(* IEC 61131-3 sources: jiepp/tests/jiepp/input, 3 files *)

(* ---- boost.iec ---- *)
{#include './boost/preprocessor/library.hpp'}
///{#include <boost/preprocessor/repetition/repeat.hpp>}
///{#include './boost/preprocessor/config/config.hpp'}

{#define DEFINE_IN_VAR(z, n, data) BOOST_PP_CAT(in, BOOST_PP_ADD(n, 1)): data;}
{#define SUM_IN_VARS(z, n, data) BOOST_PP_IF(n, +, ) BOOST_PP_CAT(in, BOOST_PP_ADD(n, 1))}

{#define DEFINE_ADD_FUNCTION(z, n, data) $
function BOOST_PP_CAT(add_, BOOST_PP_CAT(BOOST_PP_CAT(data, _), BOOST_PP_ADD(n, 2))): data $
var_input $
    BOOST_PP_REPEAT(BOOST_PP_ADD(n, 2), DEFINE_IN_VAR, data) $
end_var $
$
BOOST_PP_CAT(add_, BOOST_PP_CAT(BOOST_PP_CAT(data, _), BOOST_PP_ADD(n, 2))) := BOOST_PP_REPEAT(BOOST_PP_ADD(n, 2), SUM_IN_VARS, _); $
$
end_function $
}

BOOST_PP_REPEAT(8, DEFINE_ADD_FUNCTION, int)

{#undef SUM_IN_VARS}
{#undef DEFINE_IN_VAR}

(* ---- function_macro.iec ---- *)
{#define DECL_BIN_FUNCTION(PREFIX, OPERATOR, T) $
function PREFIX@@_@@T: T $
var_input $
	in1, in2: T; $
end_var $
$
PREFIX@@_@@T := in1 OPERATOR in2; $
$
end_function}

{#define DECL_ADD_FUNCTION(T) DECL_BIN_FUNCTION(add, +, T)}
{#define DECL_MUL_FUNCTION(T) DECL_BIN_FUNCTION(mul, *, T)}

DECL_ADD_FUNCTION(int);
DECL_MUL_FUNCTION(int);

DECL_ADD_FUNCTION(lreal);
DECL_MUL_FUNCTION(lreal);

(* ---- if.iec ---- *)
{#if true}
program Main1 __LINE__;end_program
{#endif}

{#if false}
program Main2 __LINE__;end_program
{#endif}

{#if true}
program Main3_1 __LINE__;end_program
{#else}
program Main3_2 __LINE__;end_program
{#endif}

{#if false}
program Main4_1 __LINE__;end_program
{#else}
program Main4_2 __LINE__;end_program
{#endif}

{#if false}
program Main5_1 __LINE__;end_program
{#elif false}
program Main5_2 __LINE__;end_program
{#else}
program Main5_3 __LINE__;end_program
{#endif}

{#if false}
program Main6_1 __LINE__;end_program
{#elif true}
program Main6_2 __LINE__;end_program
{#else}
program Main6_3 __LINE__;end_program
{#endif}

{#if true}
program Main7_1 __LINE__;end_program
{#elif false}
program Main7_2 __LINE__;end_program
{#else}
program Main7_3 __LINE__;end_program
{#endif}

{#if true}
program Main8_1 __LINE__;end_program
{#elif true}
program Main8_2 __LINE__;end_program
{#else}
program Main8_3 __LINE__;end_program
{#endif}
